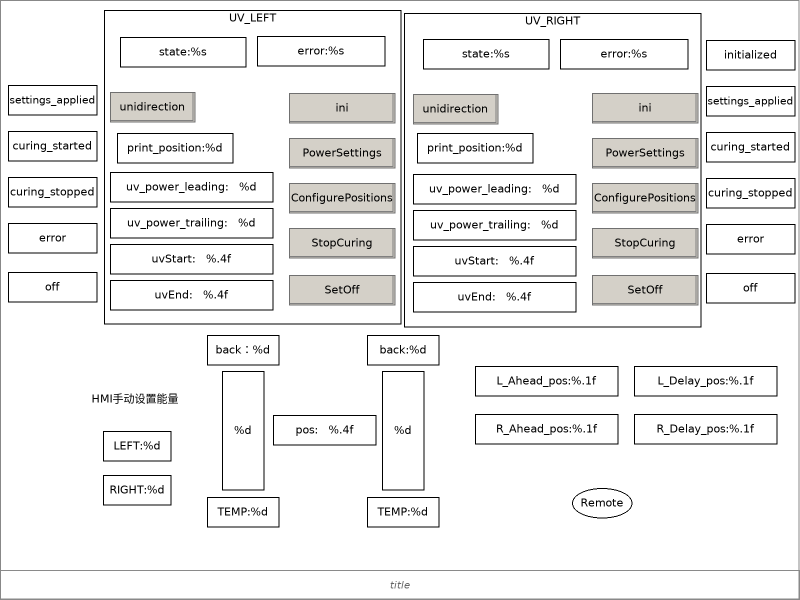
VISUALIZATION F6_UVLed  // 800x600
    RoundedRectangle (404,13 297x314), "UV_RIGHT"
    RoundedRectangle (104,10 297x314), "UV_LEFT"
    Rectangle (222,371 42x119), "%d", text variable: GVL.set_uv_power_left, colour toggle: GVL.set_uv_power_left<>0
    Rectangle (382,371 42x119), "%d", text variable: GVL.set_uv_power_right, colour toggle: GVL.set_uv_power_right<>0
    Rectangle (273,415 103x30), "pos: %.4f", text variable: Axis[1].Ref.NcToPlc.ActPos
    Button (289,93 106x30), "ini", colour toggle: GVL_API.stUVLed[1].Initialize
        toggle GVL_API.stUVLed[1].Initialize
    Rectangle (120,37 126x30), "state:%s", text list: 'TextList_UVLed_state', text index: GVL_API.stUVLed[1].state
    Rectangle (257,36 128x30), "error:%s", text list: 'TextList_UVLed_errorid', text index: GVL_API.stUVLed[1].error_code
    Rectangle (110,172 163x30), "uv_power_leading: %d", text variable: GVL_API.stUVLed[1].uv_power_leading
        OnMouseDown: write GVL_API.stUVLed[1].uv_power_leading via Default
    Button (110,92 85x30), "unidirection", colour toggle: GVL_API.stUVLed[1].unidirection
        toggle GVL_API.stUVLed[1].unidirection
    Rectangle (110,208 163x30), "uv_power_trailing: %d", text variable: GVL_API.stUVLed[1].uv_power_trailing
        OnMouseDown: write GVL_API.stUVLed[1].uv_power_trailing via Default
    Rectangle (110,244 163x30), "uvStart: %.4f", text variable: GVL_API.stUVLed[1].uvStart
        OnMouseDown: write GVL_API.stUVLed[1].uvStart via Default
    Rectangle (110,280 163x30), "uvEnd: %.4f", text variable: GVL_API.stUVLed[1].uvEnd
        OnMouseDown: write GVL_API.stUVLed[1].uvEnd via Default
    Button (289,138 106x30), "PowerSettings", colour toggle: GVL_API.stUVLed[1].ConfigurePowerSettings
        toggle GVL_API.stUVLed[1].ConfigurePowerSettings
    Button (289,275 106x30), "SetOff", colour toggle: GVL_API.stUVLed[1].SetOff
        toggle GVL_API.stUVLed[1].SetOff
    Button (289,183 106x30), "ConfigurePositions", colour toggle: GVL_API.stUVLed[1].ConfigurePositions
        toggle GVL_API.stUVLed[1].ConfigurePositions
    Button (289,228 106x30), "StopCuring", colour toggle: GVL_API.stUVLed[1].StopCuring
        toggle GVL_API.stUVLed[1].StopCuring
    Button (592,93 106x30), "ini", colour toggle: GVL_API.stUVLed[2].Initialize
        toggle GVL_API.stUVLed[2].Initialize
    Rectangle (423,39 126x30), "state:%s", text list: 'TextList_UVLed_state', text index: GVL_API.stUVLed[2].state
    Rectangle (560,39 128x30), "error:%s", text list: 'TextList_UVLed_errorid', text index: GVL_API.stUVLed[2].error_code
    Rectangle (413,174 163x30), "uv_power_leading: %d", text variable: GVL_API.stUVLed[2].uv_power_leading
        OnMouseDown: write GVL_API.stUVLed[2].uv_power_leading via Default
    Button (413,94 85x30), "unidirection", colour toggle: GVL_API.stUVLed[2].unidirection
        toggle GVL_API.stUVLed[2].unidirection
    Rectangle (413,210 163x30), "uv_power_trailing: %d", text variable: GVL_API.stUVLed[2].uv_power_trailing
        OnMouseDown: write GVL_API.stUVLed[2].uv_power_trailing via Default
    Rectangle (413,246 163x30), "uvStart: %.4f", text variable: GVL_API.stUVLed[2].uvStart
        OnMouseDown: write GVL_API.stUVLed[2].uvStart via Default
    Rectangle (413,282 163x30), "uvEnd: %.4f", text variable: GVL_API.stUVLed[2].uvEnd
        OnMouseDown: write GVL_API.stUVLed[2].uvEnd via Default
    Button (592,138 106x30), "PowerSettings", colour toggle: GVL_API.stUVLed[2].ConfigurePowerSettings
        toggle GVL_API.stUVLed[2].ConfigurePowerSettings
    Button (592,275 106x30), "SetOff", colour toggle: GVL_API.stUVLed[2].SetOff
        toggle GVL_API.stUVLed[2].SetOff
    Button (592,183 106x30), "ConfigurePositions", colour toggle: GVL_API.stUVLed[2].ConfigurePositions
        toggle GVL_API.stUVLed[2].ConfigurePositions
    Button (592,228 106x30), "StopCuring", colour toggle: GVL_API.stUVLed[2].StopCuring
        toggle GVL_API.stUVLed[2].StopCuring
    Rectangle (207,497 72x30), "TEMP:%d", text variable: GVL.HMI_TEMP_L
    Rectangle (367,497 72x30), "TEMP:%d", text variable: GVL.HMI_TEMP_R
    Rectangle (207,335 72x30), "back：%d", text variable: GVL.HMI_power_L
    Rectangle (367,335 72x30), "back:%d", text variable: GVL.HMI_power_R
    Rectangle (103,431 68x30), "LEFT:%d", text variable: PRG_SerialComm.uv_power_left_t
        OnMouseDown: toggle 
        OnMouseDown: write PRG_SerialComm.uv_power_left_t via Default
    Rectangle (103,475 68x30), "RIGHT:%d", text variable: PRG_SerialComm.uv_power_right_t
        OnMouseDown: write PRG_SerialComm.uv_power_right_t via Default
    Rectangle (417,133 116x30), "print_position:%d", text variable: GVL_API.stUVLed[2].initial_print_position
        OnMouseDown: write GVL_API.stUVLed[2].initial_print_position via Default
    Rectangle (117,133 116x30), "print_position:%d", text variable: GVL_API.stUVLed[1].initial_print_position
        OnMouseDown: write GVL_API.stUVLed[1].initial_print_position via Default
    Frame (0,570 800x30)
        shows title()
    Label (60,384 150x30), "HMI手动设置能量"
    Rectangle (475,366 143x30), "L_Ahead_pos:%.1f", text variable: GVL_API.stUVLed[1].ahead_pos
        OnMouseDown: write GVL_API.stUVLed[1].ahead_pos via Default
    Rectangle (475,414 143x30), "R_Ahead_pos:%.1f", text variable: GVL_API.stUVLed[2].ahead_pos
        OnMouseDown: write GVL_API.stUVLed[2].ahead_pos via Default
    Rectangle (634,366 143x30), "L_Delay_pos:%.1f", text variable: GVL_API.stUVLed[1].delay_pos
        OnMouseDown: write GVL_API.stUVLed[1].delay_pos via Default
    Rectangle (634,414 143x30), "R_Delay_pos:%.1f", text variable: GVL_API.stUVLed[2].delay_pos
        OnMouseDown: write GVL_API.stUVLed[2].delay_pos via Default
    Ellipse (572,488 60x30), "Remote", colour toggle: GVL.UVisRemote
    RoundedRectangle (8,85 89x30), "settings_applied", colour toggle: GVL_API.stUVLed[1].settings_applied
    RoundedRectangle (8,131 89x30), "curing_started", colour toggle: GVL_API.stUVLed[1].curing_started
    RoundedRectangle (8,223 89x30), "error", colour toggle: GVL_API.stUVLed[1].error
    RoundedRectangle (8,272 89x30), "off", colour toggle: GVL_API.stUVLed[1].off
    RoundedRectangle (8,177 89x30), "curing_stopped", colour toggle: GVL_API.stUVLed[1].curing_stopped
    RoundedRectangle (706,273 89x30), "off", colour toggle: GVL_API.stUVLed[2].off
    RoundedRectangle (706,40 89x30), "initialized", colour toggle: GVL_API.stUVLed[2].initialized
    RoundedRectangle (706,86 89x30), "settings_applied", colour toggle: GVL_API.stUVLed[2].settings_applied
    RoundedRectangle (706,132 89x30), "curing_started", colour toggle: GVL_API.stUVLed[2].curing_started
    RoundedRectangle (706,224 89x30), "error", colour toggle: GVL_API.stUVLed[2].error
    RoundedRectangle (706,178 89x30), "curing_stopped", colour toggle: GVL_API.stUVLed[2].curing_stopped
END_VISUALIZATION

(* stored: Version 1.1.0.1, ProductVersion 3.1.4024.11
   Visu F6_UVLed: Id {a4516712-de0b-467b-8638-0ad3d030056c} *)
